TYPE Read_BLPS1_Values_To_PC_Struct :
UNION
	S_BLPS1Values_To_PC:S_BLPS1Values_To_PC_Struct;
END_UNION
END_TYPE

(* stored: Version 1.1.0.1, ProductVersion 3.1.4024.16
   DUT Read_BLPS1_Values_To_PC_Struct: Id {c4448798-275e-4f71-bf01-df6f112ea13e} *)
